// TwinCAT 3 PLC project TC3_ECC203_PLC
// ProgramVersion: 3.1.4024.0
// libraries:
//   Tc2_Standard, * (Beckhoff Automation GmbH)
//   Tc2_System, * (Beckhoff Automation GmbH)
//   Tc3_Module, * (Beckhoff Automation GmbH)
// project tree:
//   DUTs/ scRCIP.TcDUT (not stored)
//   GVLs/ gRCIP.TcGVL, gCMB.TcGVL
//   / PlcTask.TcTTO
//   POUs/ MAIN.TcPOU
//   POUs/Sys/ JsonProcess.TcPOU (not stored), JsonProfile.TcPOU (not stored), PresisProcess.TcPOU (not stored), PresisProfile.TcPOU (not stored), RegProcess.TcPOU (not stored), RegProfile.TcPOU (not stored)
// real-time tasks:
//   TASK PlcTask: cycle T#10ms, priority 20, ADS port 350
// I/O:
//   DEVICE Device 1 (EtherCAT), AmsNetId 192.168.105.29.2.1
//     Box 1 (NX-ECC203) [NX-ECC203 EtherCAT coupler V1.7]

CONFIGURATION TC3_ECC203_PLC
    RESOURCE PLC ON TwinCAT3
        TASK PlcTask(INTERVAL := T#10ms, PRIORITY := 20);
        PROGRAM MAIN WITH PlcTask : MAIN;
    END_RESOURCE
END_CONFIGURATION

// ---- GVLs/gRCIP.TcGVL
{attribute 'qualified_only'}
{attribute 'pack_size' := '1'}
VAR_GLOBAL
	{region '__Chamber_Recipe_Body__' }
	RcipCMB			: ARRAY[0..100] OF scRCIP;		// Index 0 for Dummy
	{endregion}
 
	{region '__Chamber_Recipe_Profile__' }
	RcipARM			: ARRAY[0..100] OF WORD;		// Index 0 for Dummy
	{endregion}

END_VAR

// ---- GVLs/gCMB.TcGVL
{attribute 'qualified_only'}
{attribute 'pack_size' := '1'}
VAR_GLOBAL
END_VAR

// ---- POUs/MAIN.TcPOU
PROGRAM MAIN
VAR
END_VAR

END_PROGRAM
